// TIA Portal V20 export
FUNCTION_BLOCK "MotorSequenceLAD"   // FB1, LAD
{ S7_Optimized_Access := 'TRUE' }
// stored: AutoNumber true
   VAR_INPUT
      Start : Bool;
      Stop : Bool;
      StartInterval : Time;
      StopInterval : Time;
   END_VAR
   VAR_OUTPUT
      Motor1 : Bool;
      Motor2 : Bool;
      Motor3 : Bool;
      Stopping : Bool;
   END_VAR
   VAR
      Active1 : Bool;
      Active2 : Bool;
      Active3 : Bool;
      PreviousStart : Bool;
      StartPulse : Bool;
      StopEvent : Bool;
      Had3 : Bool;
      Had2 : Bool;
      Start2Done : Bool;
      Start3Done : Bool;
      Stop2Done : Bool;
      Stop1Done : Bool;
      Start2 { S7_SetPoint := 'True'} : TON_TIME;
      Start3 { S7_SetPoint := 'True'} : TON_TIME;
      Stop2 { S7_SetPoint := 'True'} : TON_TIME;
      Stop1 { S7_SetPoint := 'True'} : TON_TIME;
   END_VAR
BEGIN

REGION Network 1: 启动上升沿，仅接受新的按钮动作
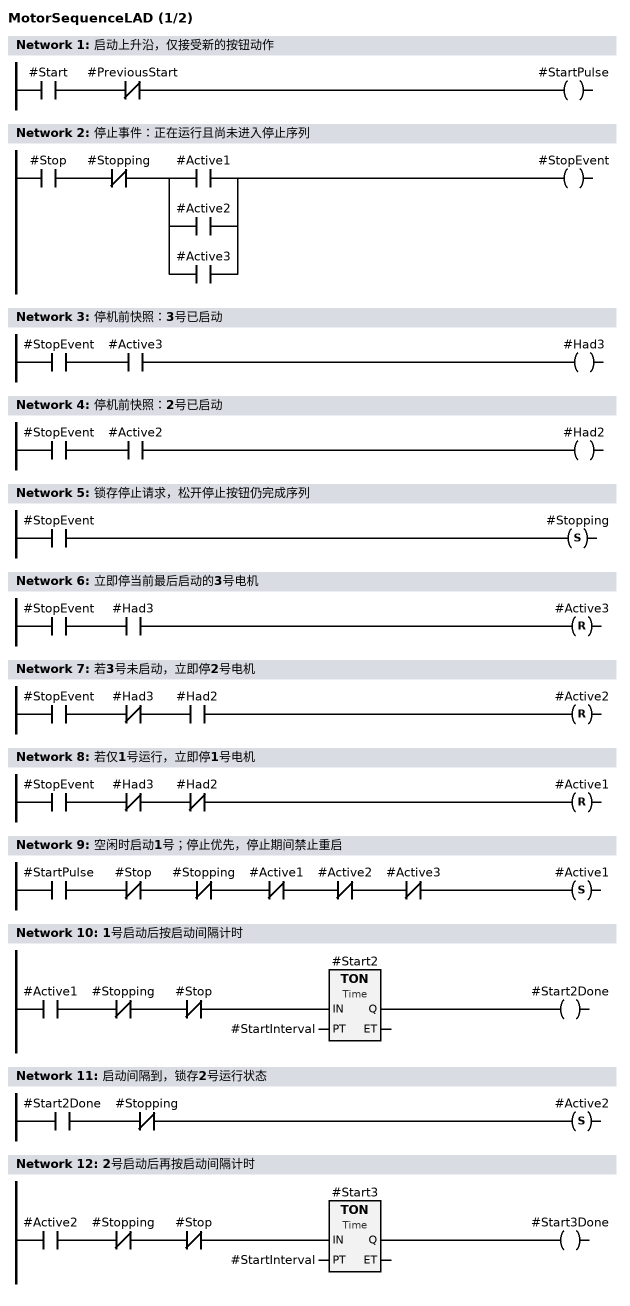
   RUNG wire#powerrail
      Contact( #Start )
      I_Contact( #PreviousStart )
      Coil( #StartPulse )
   END_RUNG
   // the same network as SCL:
   #StartPulse := #Start AND NOT #PreviousStart;
END_REGION

REGION Network 2: 停止事件：正在运行且尚未进入停止序列
   #StopEvent := #Stop AND NOT #Stopping AND (#Active1 OR #Active2 OR #Active3);
END_REGION

REGION Network 3: 停机前快照：3号已启动
   RUNG wire#powerrail
      Contact( #StopEvent )
      Contact( #Active3 )
      Coil( #Had3 )
   END_RUNG
   // the same network as SCL:
   #Had3 := #StopEvent AND #Active3;
END_REGION

REGION Network 4: 停机前快照：2号已启动
   RUNG wire#powerrail
      Contact( #StopEvent )
      Contact( #Active2 )
      Coil( #Had2 )
   END_RUNG
   // the same network as SCL:
   #Had2 := #StopEvent AND #Active2;
END_REGION

REGION Network 5: 锁存停止请求，松开停止按钮仍完成序列
   RUNG wire#powerrail
      Contact( #StopEvent )
      S_Coil( #Stopping )
   END_RUNG
   // the same network as SCL:
   IF #StopEvent THEN #Stopping := TRUE; END_IF;
END_REGION

REGION Network 6: 立即停当前最后启动的3号电机
   RUNG wire#powerrail
      Contact( #StopEvent )
      Contact( #Had3 )
      R_Coil( #Active3 )
   END_RUNG
   // the same network as SCL:
   IF #StopEvent AND #Had3 THEN #Active3 := FALSE; END_IF;
END_REGION

REGION Network 7: 若3号未启动，立即停2号电机
   RUNG wire#powerrail
      Contact( #StopEvent )
      I_Contact( #Had3 )
      Contact( #Had2 )
      R_Coil( #Active2 )
   END_RUNG
   // the same network as SCL:
   IF #StopEvent AND NOT #Had3 AND #Had2 THEN #Active2 := FALSE; END_IF;
END_REGION

REGION Network 8: 若仅1号运行，立即停1号电机
   RUNG wire#powerrail
      Contact( #StopEvent )
      I_Contact( #Had3 )
      I_Contact( #Had2 )
      R_Coil( #Active1 )
   END_RUNG
   // the same network as SCL:
   IF #StopEvent AND NOT #Had3 AND NOT #Had2 THEN #Active1 := FALSE; END_IF;
END_REGION

REGION Network 9: 空闲时启动1号；停止优先，停止期间禁止重启
   RUNG wire#powerrail
      Contact( #StartPulse )
      I_Contact( #Stop )
      I_Contact( #Stopping )
      I_Contact( #Active1 )
      I_Contact( #Active2 )
      I_Contact( #Active3 )
      S_Coil( #Active1 )
   END_RUNG
   // the same network as SCL:
   IF #StartPulse AND NOT #Stop AND NOT #Stopping AND NOT #Active1 AND NOT #Active2 AND NOT #Active3 THEN
       #Active1 := TRUE;
   END_IF;
END_REGION

REGION Network 10: 1号启动后按启动间隔计时
   RUNG wire#powerrail
      Contact( #Active1 )
      I_Contact( #Stopping )
      I_Contact( #Stop )
      { S7_Templates := "time_type := Time" } #Start2.TON(pt := #StartInterval, et =>)
      Coil( #Start2Done )
   END_RUNG
   // the same network as SCL:
   #Start2(IN := #Active1 AND NOT #Stopping AND NOT #Stop, PT := #StartInterval);   // TON
   #Start2Done := #Start2.Q;
END_REGION

REGION Network 11: 启动间隔到，锁存2号运行状态
   RUNG wire#powerrail
      Contact( #Start2Done )
      I_Contact( #Stopping )
      S_Coil( #Active2 )
   END_RUNG
   // the same network as SCL:
   IF #Start2Done AND NOT #Stopping THEN #Active2 := TRUE; END_IF;
END_REGION

REGION Network 12: 2号启动后再按启动间隔计时
   RUNG wire#powerrail
      Contact( #Active2 )
      I_Contact( #Stopping )
      I_Contact( #Stop )
      { S7_Templates := "time_type := Time" } #Start3.TON(pt := #StartInterval, et =>)
      Coil( #Start3Done )
   END_RUNG
   // the same network as SCL:
   #Start3(IN := #Active2 AND NOT #Stopping AND NOT #Stop, PT := #StartInterval);   // TON
   #Start3Done := #Start3.Q;
END_REGION

REGION Network 13: 启动间隔到，锁存3号运行状态
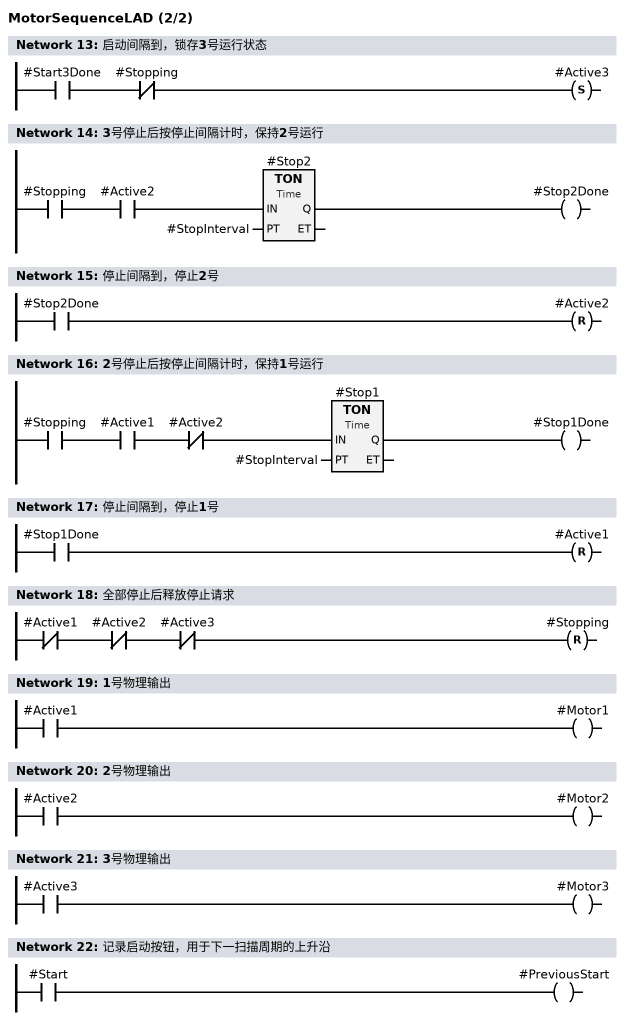
   RUNG wire#powerrail
      Contact( #Start3Done )
      I_Contact( #Stopping )
      S_Coil( #Active3 )
   END_RUNG
   // the same network as SCL:
   IF #Start3Done AND NOT #Stopping THEN #Active3 := TRUE; END_IF;
END_REGION

REGION Network 14: 3号停止后按停止间隔计时，保持2号运行
   RUNG wire#powerrail
      Contact( #Stopping )
      Contact( #Active2 )
      { S7_Templates := "time_type := Time" } #Stop2.TON(pt := #StopInterval, et =>)
      Coil( #Stop2Done )
   END_RUNG
   // the same network as SCL:
   #Stop2(IN := #Stopping AND #Active2, PT := #StopInterval);   // TON
   #Stop2Done := #Stop2.Q;
END_REGION

REGION Network 15: 停止间隔到，停止2号
   RUNG wire#powerrail
      Contact( #Stop2Done )
      R_Coil( #Active2 )
   END_RUNG
   // the same network as SCL:
   IF #Stop2Done THEN #Active2 := FALSE; END_IF;
END_REGION

REGION Network 16: 2号停止后按停止间隔计时，保持1号运行
   RUNG wire#powerrail
      Contact( #Stopping )
      Contact( #Active1 )
      I_Contact( #Active2 )
      { S7_Templates := "time_type := Time" } #Stop1.TON(pt := #StopInterval, et =>)
      Coil( #Stop1Done )
   END_RUNG
   // the same network as SCL:
   #Stop1(IN := #Stopping AND #Active1 AND NOT #Active2, PT := #StopInterval);   // TON
   #Stop1Done := #Stop1.Q;
END_REGION

REGION Network 17: 停止间隔到，停止1号
   RUNG wire#powerrail
      Contact( #Stop1Done )
      R_Coil( #Active1 )
   END_RUNG
   // the same network as SCL:
   IF #Stop1Done THEN #Active1 := FALSE; END_IF;
END_REGION

REGION Network 18: 全部停止后释放停止请求
   RUNG wire#powerrail
      I_Contact( #Active1 )
      I_Contact( #Active2 )
      I_Contact( #Active3 )
      R_Coil( #Stopping )
   END_RUNG
   // the same network as SCL:
   IF NOT #Active1 AND NOT #Active2 AND NOT #Active3 THEN #Stopping := FALSE; END_IF;
END_REGION

REGION Network 19: 1号物理输出
   RUNG wire#powerrail
      Contact( #Active1 )
      Coil( #Motor1 )
   END_RUNG
   // the same network as SCL:
   #Motor1 := #Active1;
END_REGION

REGION Network 20: 2号物理输出
   RUNG wire#powerrail
      Contact( #Active2 )
      Coil( #Motor2 )
   END_RUNG
   // the same network as SCL:
   #Motor2 := #Active2;
END_REGION

REGION Network 21: 3号物理输出
   RUNG wire#powerrail
      Contact( #Active3 )
      Coil( #Motor3 )
   END_RUNG
   // the same network as SCL:
   #Motor3 := #Active3;
END_REGION

REGION Network 22: 记录启动按钮，用于下一扫描周期的上升沿
   RUNG wire#powerrail
      Contact( #Start )
      Coil( #PreviousStart )
   END_RUNG
   // the same network as SCL:
   #PreviousStart := #Start;
END_REGION
END_FUNCTION_BLOCK
